///Get the Code from the HRESULT
FUNCTION GetCode : UINT
VAR_INPUT
    hr : HRESULT;
END_VAR
VAR
END_VAR

GetCode := UDINT_TO_UINT(DINT_TO_UDINT(hr) AND 16#0000FFFF);

END_FUNCTION

(* stored: Version 1.1.0.1, ProductVersion 3.1.4020.12
   POU GetCode: Id {8ca8ae97-dd2a-4577-b10c-49cf12ef4b3a}, SpecialFunc None *)
